{attribute addProperty BoxType "EJ7342-0000-0020"}
{attribute addProperty Id "StatusAT %I*Status_06A4ECA2162"}
{attribute addProperty CRC "1691957059"}
{attribute addProperty SizeInBites "16"}
{attribute addProperty SizeInBytes "2"}
TYPE DCM_Status_Channel_64D93743 :
STRUCT
	{attribute addProperty Name "Status"}
	Status AT %I* : Status_06A4ECA2;
END_STRUCT
END_TYPE

(* stored: Version 1.2.0.0, ProductVersion 3.1.4024.9
   DUT DCM_Status_Channel_64D93743: Id {462ccfbd-7a5a-4ec5-80c2-7b96c3ca6613} *)
